// Mitsubishi GX Works2 project: 3초씩 회전 수 증가   PLC: Q03UDV

PROGRAM MAIN
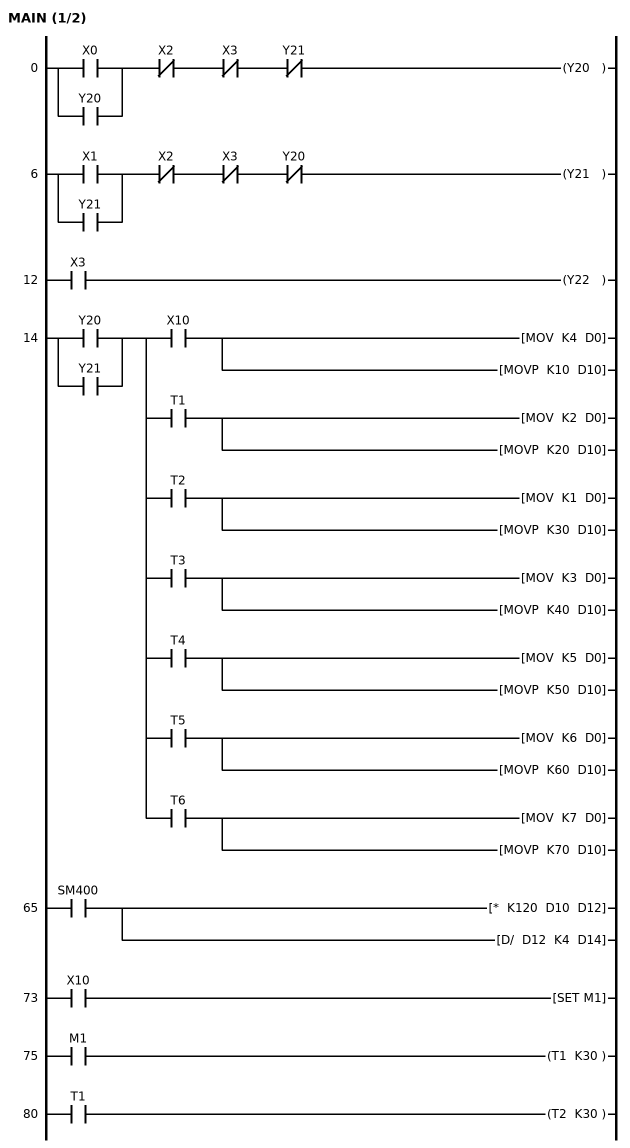
0     LD      X0
      OR      Y20
      ANI     X2
      ANI     X3
      ANI     Y21
      OUT     Y20
6     LD      X1
      OR      Y21
      ANI     X2
      ANI     X3
      ANI     Y20
      OUT     Y21
12    LD      X3
      OUT     Y22
14    LD      Y20
      OR      Y21
      MPS
      AND     X10
      MOV     K4 D0
      MOVP    K10 D10
      MRD
      AND     T1
      MOV     K2 D0
      MOVP    K20 D10
      MRD
      AND     T2
      MOV     K1 D0
      MOVP    K30 D10
      MRD
      AND     T3
      MOV     K3 D0
      MOVP    K40 D10
      MRD
      AND     T4
      MOV     K5 D0
      MOVP    K50 D10
      MRD
      AND     T5
      MOV     K6 D0
      MOVP    K60 D10
      MPP
      AND     T6
      MOV     K7 D0
      MOVP    K70 D10
65    LD      SM400
      *       K120 D10 D12
      D/      D12 K4 D14
73    LD      X10
      SET     M1
75    LD      M1
      OUT     T1 K30
80    LD      T1
      OUT     T2 K30
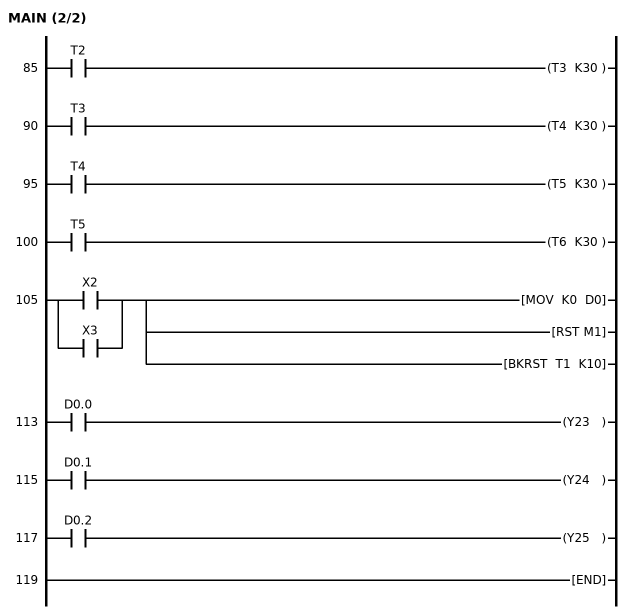
85    LD      T2
      OUT     T3 K30
90    LD      T3
      OUT     T4 K30
95    LD      T4
      OUT     T5 K30
100   LD      T5
      OUT     T6 K30
105   LD      X2
      OR      X3
      MOV     K0 D0
      RST     M1
      BKRST   T1 K10
113   LD      D0.0
      OUT     Y23
115   LD      D0.1
      OUT     Y24
117   LD      D0.2
      OUT     Y25
119   END
END_PROGRAM
